Staubli VAL3: LasMAN.dtx

bool bExit
bool bSync
bool bWelcome = true
